FUNCTION_BLOCK EcMasterConfDevices IMPLEMENTS IEcTask
VAR_INPUT
END_VAR
VAR_OUTPUT
END_VAR
VAR
	iState : INT;
	masterConfDevices : Tc2_EtherCAT.FB_EcGetConfSlaves;
	_confDevices : ARRAY[0..Tc2_EtherCAT.EC_MAX_SLAVES] OF Tc2_EtherCAT.ST_EcSlaveConfigData;
	_execute: BOOL;
	_done: BOOL;
	_busy: BOOL;	
	_error: BOOL;
	_netId: AMSNETID;
END_VAR

CASE iState OF
	0:
		IF _execute THEN
			_done := FALSE;
			_busy := TRUE;
			_error := FALSE;
			masterConfDevices.bExecute := TRUE;
			IF masterConfDevices.bBusy THEN
				iState := 10;
				_execute := FALSE;
			END_IF
		END_IF
	10:
		IF NOT masterConfDevices.bBusy THEN
			IF NOT masterConfDevices.bError THEN
				_done := TRUE;
			ELSE
				_error := TRUE;
			END_IF
			_busy := FALSE;
			masterConfDevices.bExecute := FALSE;
			iState := 0;
		END_IF
END_CASE

masterConfDevices(sNetId := Tc2_System.F_CreateAmsNetId(nIds := NetId), 
					pArrEcConfSlaveInfo := ADR(_confDevices), 
					cbBufLen := SIZEOF(_confDevices));

{warning 'add method implementation '}
METHOD Abort : BOOL
masterConfDevices.bExecute := FALSE;
_busy := FALSE;
_execute := FALSE;
Abort := TRUE;
iState := 0;
END_METHOD

{warning 'add property implementation'}
PROPERTY Busy : BOOL
GET
Busy := _busy;
END_GET
END_PROPERTY

PROPERTY ConfiguredDevices : reference to array[0..Ec_Max_slaves] of St_ecslaveconfigdata
GET
ConfiguredDevices REF= _confDevices;
END_GET
END_PROPERTY

{warning 'add property implementation'}
PROPERTY Done : BOOL
GET
Done := _done;
END_GET
END_PROPERTY

{warning 'add property implementation'}
PROPERTY Error : BOOL
GET
Error := _error;
END_GET
END_PROPERTY

{warning 'add method implementation '}
METHOD Execute : BOOL
IF NOT masterConfDevices.bBusy THEN
	Execute := _execute := true;
END_IF
END_METHOD

{warning 'add property implementation'}
PROPERTY NetID : amsnetid
GET
NetID := _netId;
END_GET
SET
_netId := NetID;
END_SET
END_PROPERTY

PROPERTY NumberConfDevices : udint
GET
NumberConfDevices := masterConfDevices.nSlaves;
END_GET
END_PROPERTY

END_FUNCTION_BLOCK

(* stored: Version 1.1.0.1, ProductVersion 3.1.4024.9
   POU EcMasterConfDevices: Id {bfb15777-5ac2-47f5-997a-05d929608a62}, SpecialFunc None
   Method Abort: Id {7b340730-3588-40ad-a653-fa5775c54f50}
   Property Busy: Id {a4575f44-7364-49f4-9d7a-2ee9f4166947}
   Get Get: Id {1e725270-54ff-411c-a5e7-6193a67f91a4}
   Property ConfiguredDevices: Id {d7ab2219-abed-40ed-9b3e-2b1d3829f83e}
   Get Get: Id {934f027a-85c7-41df-aff3-e6ccfc7af7fc}
   Property Done: Id {bfcb367e-1477-4e86-8f1b-4e573c57198e}
   Get Get: Id {39832905-f539-4b41-8360-65532f044f7b}
   Property Error: Id {dc845e02-a0f3-4212-8f21-6e6cd3c07990}
   Get Get: Id {de8a3733-cfc4-4578-b02f-218ca6d7e370}
   Method Execute: Id {d9d7bf50-43f4-43f0-a288-bdc9c2669ecc}
   Property NetID: Id {383db7e8-627b-46f8-8f1d-f51ee527446c}
   Get Get: Id {7aa91ba4-338a-4523-b1a5-11eacb7c732d}
   Set Set: Id {768d3337-4c06-4d35-8880-9f9d38f929b9}
   Property NumberConfDevices: Id {11f59a4d-6251-402e-9bb1-feed57c6b0b4}
   Get Get: Id {172cc73d-5e90-4b62-80e2-80e65e56b1ff} *)
